# EPICS substitutions: modules/event/evrSupport/Db/ioc/IOC-IN20-MG01evr.substitutions
#==============================================================================
#
# Abs:  LCLS EVR IOC records for IN20 MG01
#
# Name: IOC-IN20-MG01evr.substitutions
#
#==============================================================================
#
file evrMGXX.db
{
pattern { DEVICE        }
	{ EVR:IN20:MG01 }
}
